Staubli VAL3: getFrame.pgx

public program getFrame(frame& x_fFrame[], bool x_bCycle)
  local num l_nIndex
begin
  // CYCLE
  if x_bCycle
    l_nIndex=pt:tTraj[sTrajCycle].nIndexFrame
  else
    // NOT CYCLE
    l_nIndex=jEditPoint.nIndexFrame
  endIf
  x_fFrame.trsf=saveData:fFrameItem[l_nIndex].fFrame.trsf
end
